Staubli VAL3: Custom.pjx

--- Custom.pjx ---
Parameters version=s7.7 stackSize=5000 millimeterUnit=true
Program file=AfterArrayCut.pgx
Program file=AfterCloseLaser.pgx
Program file=AfterOpenLaser.pgx
Program file=AfterProduct.pgx
Program file=AfterTraj.pgx
Program file=AfterWorkPlace.pgx
Program file=BeforeAppro.pgx
Program file=BeforeArrayCut.pgx
Program file=BeforeCut.pgx
Program file=BeforeOpenLaser.pgx
Program file=BeforeProduct.pgx
Program file=BeforeTraj.pgx
Program file=ChooseCustomPro.pgx
Program file=CustomPoll.pgx
Program file=ReadMe.pgx
Program file=start.pgx
Program file=stop.pgx
Data file=Custom.dtx

--- Custom.dtx ---
mdesc mNomSpeed
bool bDebug
dio dAlarm = {link=ModbusSrv-0\Modbus-Bit\UsIn_bNull1}
dio dSafety1 = {link=ModbusSrv-0\Modbus-Bit\In2_bNull2}
dio dSafety2 = {link=ModbusSrv-0\Modbus-Bit\UsIn_bNull3}
dio dSaftey3 = {link=ModbusSrv-0\Modbus-Bit\UsIn_bNull3}
dio dSaftey4 = {link=ModbusSrv-0\Modbus-Bit\UsO_bNull5}
dio dSation1
dio dSation2
dio dSation3
dio dSation4

--- AfterArrayCut.pgx ---
public program AfterArrayCut(num x_nTrajIndex)
begin
  //在阵列之后添加动作








end

--- AfterCloseLaser.pgx ---
public program AfterCloseLaser()
begin
  //激光关闭以后需要做的动作
  //离开点还没有运行之前
  //在motion.pjx中的move.pgx中
  //请使用ctr+F进行全局查找



end

--- AfterOpenLaser.pgx ---
public program AfterOpenLaser()
begin
  //激光打开以后需要做的动作
  //机械手臂在穿孔的时候
  //在motion.pjx中的move.pgx中
  //请使用ctr+F进行全局查找




end

--- AfterProduct.pgx ---
public program AfterProduct(num x_nWorkplaceIn)
  local num l_nNum
begin
  //产品生产之后需要进行的工作
  //路径完成，但是没有回零
  //外部轴也没有进行归位
  //与AfterWorkPlace区别是AfterWorkPlace机械手臂回到零位
  //如果要加信号，请在前面加上waitendmove()
























//  //路径过滤的话
//  //启动时把下面的话语注释掉
//
//  if TxtFile:bTrajFilter
//    for l_nNum=0 to TxtFile:nTotalTraj-1
//
//      TxtFile:bBypass[l_nNum]=false
//
//    endFor
//
//    call TrajByPass(1,TxtFile:nTotalTraj)
//
//  endIf




//添加



end

--- AfterTraj.pgx ---
public program AfterTraj(num x_nTrajIndex)
begin
   //在motion.pjx中的move.pgx中
  //请使用ctr+F进行全局查找
  //用在完成离开点之后
  //添加动作需要waitendmove()


//
//    if bDebug
//    popUpMsg("AfterTraj")
//    logMsg("AfterTraj")
//
//
//    endIf






















end

--- AfterWorkPlace.pgx ---
public program AfterWorkPlace(num x_nIndex)
begin
  //工位完成后，可以输出IO
  //


//  if bDebug
//    popUpMsg("AfterWorkPlace")
//    logMsg("AfterWorkPlace")
//
//
//  endIf



end

--- BeforeAppro.pgx ---
public program BeforeAppro()
begin
  //在motion.pjx中的move.pgx中
  //请使用ctr+F进行全局查找
  //用在趋近点第一点之前



//
//  if bDebug
//    popUpMsg("BeforeAppro")
//    logMsg("BeforeAppro")
//
//
//  endIf









end

--- BeforeArrayCut.pgx ---
public program BeforeArrayCut(num x_nTrajindex)
begin
  //在阵列之前添加动作





end

--- BeforeCut.pgx ---
public program BeforeCut()
begin

  //在穿孔点之前的函数
  //可以添加需要的内容















end

--- BeforeOpenLaser.pgx ---
public program BeforeOpenLaser()
begin
  //在motion.pjx中的move.pgx中
  //请使用ctr+F进行全局查找
  //用在切割点开光之前
  //


//  if bDebug
//    popUpMsg("beforelaser")
//    logMsg("beforelaser")
//
//
//  endIf







end

--- BeforeProduct.pgx ---
public program BeforeProduct(num x_nWorkPlaceIn)
  local num l_nNum
begin
  //产品开始生产前所需要做的工作
  //安全信号的确认之类


















  //路径过滤的话
  //启动时把下面的话语注释掉

//  if TxtFile:bTrajFilter
//    for l_nNum=0 to TxtFile:nTotalTraj-1
//
//      TxtFile:bBypass[l_nNum]=false
//
//    endFor
//
//    call TrajByPass(1,TxtFile:nTotalTraj)
//
//  endIf


end

--- BeforeTraj.pgx ---
public program BeforeTraj(num x_nTrajIndex)
begin

  //调用位置在Motion库中Move函数中
  //用在路径开始之前


   //

//   if bDebug
//
//
//
//
//
//
//  endIf



end

--- ChooseCustomPro.pgx ---
public program ChooseCustomPro(num& x_nWorkplace, num& x_nProductIndex)
begin
  //对应客户自定义方式来选择相对应的产品
  //在触发方式中 有客户自定义触发
  //2014.06.03

//  x_nWorkplace=0
//  while x_nWorkplace==0
//
//    if bDebug
//      if dSafety1==true and dSation1==true
//        x_nWorkplace=1
//      endIf
//
//
//      if dSafety2==true and dSation2==true
//        x_nWorkplace=2
//      endIf
//
//      if dSaftey3==true and dSation3==true
//        x_nWorkplace=3
//      endIf
//
//      if dSaftey4==true and dSation4==true
//        x_nWorkplace=4
//      endIf
//
//
//    endIf
//
//
//
//    delay(0)
//  endWhile






end

--- CustomPoll.pgx ---
public program CustomPoll()
  local num l_nNum
begin
  //用户在轮询函数中添加自己需要检查的内容
  //  可以添加报警信号
  //如果报警，则下电 dispower()
  //logmess


//  if dAlarm==true
//    disablePower()
//    logMsg("aAlarm 报警触发")
//
//  endIf






end

--- ReadMe.pgx ---
public program ReadMe()
begin
  //这是一个提供给客户的自定义开发的程序
  //这个库不引用其他库
  //这个库里面的界面，IO都是在这个库里面自己定义。
  //
  //注意相应的逻辑顺序
  //客户应该具有VAL3熟练编程能力，知道编程逻辑，理解代码能力
  //库中已经提供好函数名称与函数的参数，只需要对相应的参数进行定义就好了



















end
